FUNCTION_BLOCK fb_testpiston
VAR_INPUT
END_VAR
VAR_OUTPUT
END_VAR
VAR
	step: INT;
	wait1: TON;
	wait2: TON;
	unlock: INT;
	failUp: INT;
	failDown: INT;
	lock: INT;
	wait: INT;
	totalFail: INT;
	wait3: TON;
	wait4: TON;
END_VAR

IF (unlock > 50 AND lock > 50) OR totalFail <> 0 THEN
	ADSLOGDINT( msgCtrlMask := ADSLOG_MSGTYPE_HINT OR ADSLOG_MSGTYPE_MSGBOX, 
                    msgFmtStr := 'test Msg: Test DONE! Number of fails: %d', dintArg:= totalFail);
	ADSLOGDINT( msgCtrlMask := ADSLOG_MSGTYPE_HINT OR ADSLOG_MSGTYPE_MSGBOX, 
                    msgFmtStr := '%d Unlock fails', dintArg:= failUp);
	ADSLOGDINT( msgCtrlMask := ADSLOG_MSGTYPE_HINT OR ADSLOG_MSGTYPE_MSGBOX, 
                    msgFmtStr := '%d Lock fails', dintArg:= failDown);
	wait1.IN := FALSE;
	wait2.IN := FALSE;
	unlock := 0;
	lock := 0;
	totalFail := 0;
	failDown := 0;
	failUp := 0;
	step := 1000;
END_IF

CASE step OF
	0: 
		step := 10;
	10:
		wait3(IN := TRUE, PT := T#1000MS);
		IF tcin.ProxUp THEN
			IF wait3.Q THEN
				wait2.IN := FALSE;
				wait3.IN := FALSE;
				tcout.valvePush := TRUE;
				tcout.valvePull := FALSE;
				wait1(IN := TRUE, PT := T#10S);
				step := 20;
				unlock := unlock + 1;
			END_IF
		ELSIF wait2.Q THEN
			step := 991;
		END_IF
		
	20:
		wait4(IN := TRUE, PT := T#1000MS);
		IF tcin.ProxDwn THEN
			IF wait4.Q THEN
				wait4.IN := FALSE;
				wait1.IN := FALSE;
				tcout.valvePull := TRUE;
				tcout.valvePush := FALSE;
				wait2(IN := TRUE, PT := T#10S);
				step := 10;
				lock := lock + 1;
			END_IF
		ELSIF wait1.Q THEN
			step := 992;
		END_IF
		
	991:
		failUp := failUp + 1;
		step := 999;
		
	992:
		failDown := failDown + 1;
		step := 999;
		
	999:
		totalFail := totalFail + 1;
		wait1.IN := FALSE;
		wait2.IN := FALSE;
		step := 1001;
	
	1000:
		step := 0;
		
	1001:
		
END_CASE
wait4();
wait3();
wait2();
wait1();

END_FUNCTION_BLOCK

(* stored: Version 1.1.0.1, ProductVersion 3.1.4024.5
   POU fb_testpiston: Id {c5a1407f-0b88-4b83-8264-7b98061fcada}, SpecialFunc None *)
